TYPE ST_SlaveStatus :
STRUCT
	
	// state machine
	m_armState:ARRAY[1..g_sArmNum] OF E_SlaveArmState;
	
	// instrument info
	m_instruStauts :ARRAY[1..g_sArmNum] OF ST_InstruStatus;
	
	// command arm pose in endoscope view
	m_cmdArmPose:ARRAY[1..g_sArmNum] OF ST_Frame;
	
	// current arm pose in endoscope view
	m_curArmPose:ARRAY[1..g_sArmNum] OF ST_Frame;
	
	// command arm twist[linear velocity; angular veloicty] in endoscope view
	m_cmdArmTwist:ARRAY[1..g_sArmNum,1..6] OF LREAL;
	
	// current arm twist[linear velocity; angular veloicty] in endoscope view
	m_curdArmTwist:ARRAY[1..g_sArmNum,1..6] OF LREAL;
	
	// joint position compute with motor encoder
	m_curMotorPos :ARRAY[1..g_sArmNum, 1..g_sJntNum] OF LREAL;
	
	// joint position compute with link/abs encoder
	m_curLinkPos :ARRAY[1..g_sArmNum, 1..g_sJntNum] OF LREAL;
	
	// target joint position 
	m_cmdJntPos :ARRAY[1..g_sArmNum, 1..g_sJntNum] OF LREAL;
	
	// current joint position 
	m_curJntPos :ARRAY[1..g_sArmNum, 1..g_sJntNum] OF LREAL;
	
	// target joint velocity 
	m_cmdJntVel :ARRAY[1..g_sArmNum, 1..g_sJntNum] OF LREAL;
	
	// current joint position 
	m_curJntVel :ARRAY[1..g_sArmNum, 1..g_sJntNum] OF LREAL;
	
	// command joint torque 
	m_cmdJntTrq :ARRAY[1..g_sArmNum, 1..g_sJntNum] OF LREAL;
	
	// current joint torque 
	m_curJntTrq :ARRAY[1..g_sArmNum, 1..g_sJntNum] OF LREAL;
END_STRUCT
END_TYPE

(* stored: Version 1.1.0.1, ProductVersion 3.1.4024.12
   DUT ST_SlaveStatus: Id {8673ecde-c145-4df2-8157-2e6da5d46538} *)
